// TwinCAT 3 PLC project MonetRoofTests
// Title: MonetRoofTests
// Company: BROT
// ProjectVersion: 0.1.0
// ProgramVersion: 3.1.4024.66
// libraries:
//   MONET Roof, * (Georg-August-Universitaet Goettingen)
//   BROTLib, * (BROT)
//   Tc2_Standard, * (Beckhoff Automation GmbH)
//   Tc2_System, * (Beckhoff Automation GmbH)
//   Tc2_Utilities, * (Beckhoff Automation GmbH)
//   Tc3_Module, * (Beckhoff Automation GmbH)
//   TcUnit, * (www.tcunit.org)
// project tree:
//   / PlcTask.TcTTO
//   POUs/ FB_NullComm.TcPOU, FB_Ramp_Tests.TcPOU, FB_Roof_Consistency_Tests.TcPOU, FB_Roof_State_Tests.TcPOU, MAIN.TcPOU
// real-time tasks:
//   TASK PlcTask: cycle T#10ms, priority 20, ADS port 350

CONFIGURATION MonetRoofTests
    RESOURCE PLC ON TwinCAT3
        TASK PlcTask(INTERVAL := T#10ms, PRIORITY := 20);
        PROGRAM MAIN WITH PlcTask : MAIN;
    END_RESOURCE
END_CONFIGURATION

// ---- POUs/MAIN.TcPOU
PROGRAM MAIN
VAR
	// TcUnit finds every FB_TestSuite instance by itself; it is enough to declare them here.
	fbRampTests				: FB_Ramp_Tests;
	fbRoofConsistencyTests	: FB_Roof_Consistency_Tests;
	fbRoofStateTests		: FB_Roof_State_Tests;
END_VAR

TcUnit.RUN();

END_PROGRAM

// ---- POUs/FB_Ramp_Tests.TcPOU
// Tests for MONETRoof.FB_Ramp, the per-call velocity ramp.
//
// FB_Ramp holds no state of its own: every call recomputes `value` fresh from the `start` input, so
// a multi-cycle ramp only happens because the caller (FB_Roof) feeds its own persisted speed back in
// as `start` each cycle. All these tests can therefore drive a fresh instance directly within a
// single method call, calling it as many times as needed in a FOR loop.
FUNCTION_BLOCK FB_Ramp_Tests EXTENDS TcUnit.FB_TestSuite
VAR
END_VAR

Single_Step_Increases_Toward_Target();
Single_Step_Decreases_Toward_Target();
Reaches_Target_Without_Overshoot();
Reaches_Target_Without_Undershoot();
Large_Reversal_Steps_Instead_Of_Jumping();
Full_Reversal_Ramps_Through_Zero_Over_Many_Cycles();
Zero_Accel_Never_Moves();

METHOD PRIVATE Single_Step_Increases_Toward_Target
VAR
	fbRamp	: MONETRoof.FB_Ramp;
END_VAR
TEST('Single_Step_Increases_Toward_Target');
fbRamp(start := 0, target := 1000, accel := 100);
AssertEquals_INT(Expected := 100, Actual := fbRamp.value, Message := 'one step of 100 towards +1000');
TEST_FINISHED();
END_METHOD

METHOD PRIVATE Single_Step_Decreases_Toward_Target
VAR
	fbRamp	: MONETRoof.FB_Ramp;
END_VAR
TEST('Single_Step_Decreases_Toward_Target');
fbRamp(start := 1000, target := 0, accel := 100);
AssertEquals_INT(Expected := 900, Actual := fbRamp.value, Message := 'one step of 100 towards 0');
TEST_FINISHED();
END_METHOD

METHOD PRIVATE Reaches_Target_Without_Overshoot
VAR
	fbRamp	: MONETRoof.FB_Ramp;
END_VAR
TEST('Reaches_Target_Without_Overshoot');
// 950 + 100 would be 1050: must clamp to the target instead
fbRamp(start := 950, target := 1000, accel := 100);
AssertEquals_INT(Expected := 1000, Actual := fbRamp.value, Message := 'clamped at target, not 1050');
TEST_FINISHED();
END_METHOD

METHOD PRIVATE Reaches_Target_Without_Undershoot
VAR
	fbRamp	: MONETRoof.FB_Ramp;
END_VAR
TEST('Reaches_Target_Without_Undershoot');
// 50 - 100 would be -50: must clamp to the target instead
fbRamp(start := 50, target := 0, accel := 100);
AssertEquals_INT(Expected := 0, Actual := fbRamp.value, Message := 'clamped at target, not -50');
TEST_FINISHED();
END_METHOD

METHOD PRIVATE Large_Reversal_Steps_Instead_Of_Jumping
VAR
	fbRamp	: MONETRoof.FB_Ramp;
END_VAR
// Regression test for code review finding H1: target - value on two INTs overflowed 16 bit for a
// reversal like -30000 -> +30000 (60000 does not fit), which flipped the sign of the comparison and
// jumped straight to the target in one step (fixed by computing it in DINT, FB_Ramp.TcPOU:19-20).
// This asserts one ramp step, not the jump the old code produced.
TEST('Large_Reversal_Steps_Instead_Of_Jumping');
fbRamp(start := -30000, target := 30000, accel := 150);
AssertEquals_INT(Expected := -29850, Actual := fbRamp.value, Message := '-30000 -> +30000: one step of 150, not a jump to +30000');
// symmetric: the same reversal the other way round
fbRamp(start := 30000, target := -30000, accel := 150);
AssertEquals_INT(Expected := 29850, Actual := fbRamp.value, Message := '+30000 -> -30000: one step of 150, not a jump to -30000');
TEST_FINISHED();
END_METHOD

METHOD PRIVATE Full_Reversal_Ramps_Through_Zero_Over_Many_Cycles
VAR
	fbRamp			: MONETRoof.FB_Ramp;
	i				: INT;
	prevValue		: INT;
	curValue		: INT;
	bAllStepsBounded	: BOOL := TRUE;
	valueAtStep200	: INT;
END_VAR
// Drives a full -30000 -> +30000 reversal the way FB_Roof does (feeding value back in as the next
// call's start) and checks every intermediate step, not just the first one. -30000 + 200*150 = 0
// exactly, so this also confirms the ramp actually passes through zero at a known step, not just
// that the endpoints are right. Uses local flags instead of one assertion per loop iteration: TcUnit
// budgets asserts per suite (256 here), and this alone would be 400 calls.
TEST('Full_Reversal_Ramps_Through_Zero_Over_Many_Cycles');
curValue := -30000;
FOR i := 1 TO 400 DO
	prevValue := curValue;
	fbRamp(start := prevValue, target := 30000, accel := 150);
	curValue := fbRamp.value;
	IF ABS(TO_DINT(curValue) - TO_DINT(prevValue)) > 150 THEN
		bAllStepsBounded := FALSE;
	END_IF
	IF i = 200 THEN
		valueAtStep200 := curValue;
	END_IF
END_FOR
AssertTrue(Condition := bAllStepsBounded, Message := 'no single step exceeded accel (150)');
AssertEquals_INT(Expected := 0, Actual := valueAtStep200, Message := 'passes through exactly 0 at step 200 (-30000 + 200*150)');
AssertEquals_INT(Expected := 30000, Actual := curValue, Message := 'reaches target after 400 steps of 150 (60000 / 150)');
TEST_FINISHED();
END_METHOD

METHOD PRIVATE Zero_Accel_Never_Moves
VAR
	fbRamp	: MONETRoof.FB_Ramp;
END_VAR
// accel = 0 is one of the config_error conditions FB_Roof guards against (M0/L6); documented here as
// what FB_Ramp itself does with it, in isolation: it never reaches the target.
TEST('Zero_Accel_Never_Moves');
fbRamp(start := 100, target := 1000, accel := 0);
AssertEquals_INT(Expected := 100, Actual := fbRamp.value, Message := 'accel = 0: value never leaves start');
TEST_FINISHED();
END_METHOD

END_FUNCTION_BLOCK

// ---- POUs/FB_Roof_Consistency_Tests.TcPOU
// Tests for MONETRoof.FB_Roof's consistency checks: sync_error, overtravel_error, config_error (code
// review findings M1, M7 and L6).
//
// TwinCAT only allows external code to WRITE a VAR_INPUT of another instance; a VAR_OUTPUT (even one
// with no AT clause) is read-only from outside, and a plain VAR (no AT/INPUT/OUTPUT) is not reachable
// at all -- only calling a public METHOD on it is. That shapes what these tests can drive:
//   - motors[i].SetPosition(x) works: it is a public METHOD, called on FB_Roof's private motors array
//     element, and is how FB_Roof itself sets a position on a limit snap.
//   - motors[i].position_open / .position_close cannot be written directly (plain VAR_OUTPUT, no
//     setter) -- so limit_error's positive case (a drive that overran its own switch) is not covered
//     here: it needs position_open, which is only ever set by the opened/closed edge, both AT%I*.
//   - position_valid cannot be written directly either (VAR_OUTPUT PERSISTENT, no setter) -- so
//     overtravel_error's positive case is not covered; the negative case (no overtravel_error while
//     position_valid is FALSE, its default) is, since that only needs a read.
// Validate limit_error and overtravel_error's positive cases on the real roof, or with I/O linked in
// a project that has it (MONETN, MONETS) -- same limitation as FB_Roof_State_Tests' opened/closed.
//
// comm is BROTLib.I_Comm, not the roof interface: an unassigned (null) reference would fault the PLC
// the first time an error/state edge tries to log through it, so every roof instance below is given
// an FB_NullComm.
FUNCTION_BLOCK FB_Roof_Consistency_Tests EXTENDS TcUnit.FB_TestSuite
VAR
END_VAR

Sync_Error_When_Positions_Differ_By_Threshold_Or_More();
Sync_Error_Clears_When_Positions_Converge();
No_Overtravel_Error_When_Position_Not_Valid();
Config_Error_When_Max_Position_Not_Above_Min();
Config_Error_When_Speed_Invalid();
Config_Error_Holds_Roof_At_Zero_Speed();

// Shared call with fixed speed/position parameters (10000/30000/150, 0..200), only max_position_diff
// varies per test. Tests that need a different min_position/max_position/speed call fbRoof directly.
METHOD PRIVATE Call
VAR_IN_OUT
	roof		: MONETRoof.FB_Roof;
END_VAR
VAR_INPUT
	comm		: BROTLib.I_Comm;
	maxPosDiff	: INT := 2;
END_VAR
roof(
	roof_number			:= 1,
	min_speed			:= 10000,
	max_speed			:= 30000,
	acceleration		:= 150,
	min_position		:= 0,
	max_position		:= 200,
	max_position_diff	:= maxPosDiff,
	comm				:= comm);
END_METHOD

METHOD PRIVATE Sync_Error_When_Positions_Differ_By_Threshold_Or_More
VAR
	fbRoof	: MONETRoof.FB_Roof;
	fbComm	: FB_NullComm;
END_VAR
TEST('Sync_Error_When_Positions_Differ_By_Threshold_Or_More');
Call(roof := fbRoof, comm := fbComm, maxPosDiff := 2);
AssertFalse(Condition := fbRoof.sync_error, Message := 'both motors start at position 0: in sync');
fbRoof.motors[1].SetPosition(100);
fbRoof.motors[2].SetPosition(102);
Call(roof := fbRoof, comm := fbComm, maxPosDiff := 2);
AssertTrue(Condition := fbRoof.sync_error, Message := 'a difference of 2 (>= max_position_diff) trips sync_error');
TEST_FINISHED();
END_METHOD

METHOD PRIVATE Sync_Error_Clears_When_Positions_Converge
VAR
	fbRoof	: MONETRoof.FB_Roof;
	fbComm	: FB_NullComm;
END_VAR
TEST('Sync_Error_Clears_When_Positions_Converge');
Call(roof := fbRoof, comm := fbComm, maxPosDiff := 2);
fbRoof.motors[1].SetPosition(100);
fbRoof.motors[2].SetPosition(101);
Call(roof := fbRoof, comm := fbComm, maxPosDiff := 2);
AssertFalse(Condition := fbRoof.sync_error, Message := 'a difference of 1 stays below the threshold of 2');
TEST_FINISHED();
END_METHOD

METHOD PRIVATE No_Overtravel_Error_When_Position_Not_Valid
VAR
	fbRoof	: MONETRoof.FB_Roof;
	fbComm	: FB_NullComm;
END_VAR
// M7: position_valid is forced FALSE on the very first cycle and only a limit snap sets it TRUE
// again, so a fresh/unconfirmed position must not arm overtravel_error even when it is wildly off.
TEST('No_Overtravel_Error_When_Position_Not_Valid');
Call(roof := fbRoof, comm := fbComm, maxPosDiff := 2);
AssertFalse(Condition := fbRoof.position_valid, Message := 'position_valid starts FALSE: never confirmed by a limit snap');
fbRoof.Open();
Call(roof := fbRoof, comm := fbComm, maxPosDiff := 2);
fbRoof.motors[1].SetPosition(500);
Call(roof := fbRoof, comm := fbComm, maxPosDiff := 2);
AssertFalse(Condition := fbRoof.overtravel_error, Message := 'no overtravel_error without position_valid, however far off the position is');
TEST_FINISHED();
END_METHOD

METHOD PRIVATE Config_Error_When_Max_Position_Not_Above_Min
VAR
	fbRoof	: MONETRoof.FB_Roof;
	fbComm	: FB_NullComm;
END_VAR
TEST('Config_Error_When_Max_Position_Not_Above_Min');
fbRoof(roof_number := 1, min_speed := 10000, max_speed := 30000, acceleration := 150,
	min_position := 100, max_position := 100, max_position_diff := 2, comm := fbComm);
AssertTrue(Condition := fbRoof.config_error, Message := 'max_position (100) not above min_position (100)');
AssertTrue(Condition := fbRoof.state = E_RoofState.error, Message := 'config_error puts the roof into the error state');
TEST_FINISHED();
END_METHOD

METHOD PRIVATE Config_Error_When_Speed_Invalid
VAR
	fbRoof	: MONETRoof.FB_Roof;
	fbComm	: FB_NullComm;
END_VAR
TEST('Config_Error_When_Speed_Invalid');
fbRoof(roof_number := 1, min_speed := 30000, max_speed := 10000, acceleration := 150,
	min_position := 0, max_position := 200, max_position_diff := 2, comm := fbComm);
AssertTrue(Condition := fbRoof.config_error, Message := 'min_speed (30000) above max_speed (10000)');
TEST_FINISHED();
END_METHOD

METHOD PRIVATE Config_Error_Holds_Roof_At_Zero_Speed
VAR
	fbRoof	: MONETRoof.FB_Roof;
	fbComm	: FB_NullComm;
END_VAR
// L1/config_error interaction: a roof already moving that picks up an invalid parameter (e.g. a
// max_speed above 32767, which would wrap TO_INT and could reverse the direction) must be held at
// zero immediately, unconditionally -- not just flagged.
TEST('Config_Error_Holds_Roof_At_Zero_Speed');
Call(roof := fbRoof, comm := fbComm, maxPosDiff := 2);
fbRoof.Open();
Call(roof := fbRoof, comm := fbComm, maxPosDiff := 2);
AssertFalse(Condition := fbRoof.config_error, Message := 'valid parameters so far');
fbRoof(roof_number := 1, min_speed := 10000, max_speed := 40000, acceleration := 150,
	min_position := 0, max_position := 200, max_position_diff := 2, comm := fbComm);
AssertTrue(Condition := fbRoof.config_error, Message := 'max_speed above 32767 wraps TO_INT: config_error catches it');
AssertTrue(Condition := fbRoof.state = E_RoofState.error, Message := 'error state; drive held, slow mode included (FB_Roof.TcPOU config_error stop)');
TEST_FINISHED();
END_METHOD

END_FUNCTION_BLOCK

// ---- POUs/FB_NullComm.TcPOU
// No-op I_Comm implementation for tests. FB_Roof/FB_RoofMotor call Comm.Publish / Comm.PublishLog
// (via FB_EventLog) on error/state edges; a null (unassigned) I_Comm reference there would fault the
// PLC, so every FB_Roof test instance is given one of these instead of a real MQTT connection.
FUNCTION_BLOCK FB_NullComm IMPLEMENTS BROTLib.I_Comm
VAR
	// number of Publish/PublishLog calls seen, in case a test ever wants to assert an event fired
	nPublishCalls		: UDINT;
	nPublishLogCalls	: UDINT;
END_VAR

METHOD Publish : BOOL
VAR_INPUT
	domain			: STRING(255) := 'environment';
	location		: STRING(255) := 'roof';
	parameter		: STRING(255);
	value			: STRING(255);
END_VAR
VAR_OUTPUT
	published	: BOOL;
END_VAR
nPublishCalls := nPublishCalls + 1;
published := TRUE;
Publish := TRUE;
END_METHOD

METHOD PublishLog : BOOL
VAR_INPUT
	level		: STRING(255) := 'INFO';
	message		: STRING(255);
END_VAR
VAR_OUTPUT
	published	: BOOL;
END_VAR
nPublishLogCalls := nPublishLogCalls + 1;
published := TRUE;
PublishLog := TRUE;
END_METHOD

END_FUNCTION_BLOCK

// ---- POUs/FB_Roof_State_Tests.TcPOU
// Tests for MONETRoof.FB_Roof's state machine (code review finding L5): the E_RoofState.unknown default
// before the first call, and what the roof does while a drive reports an error.
//
// In this project every drive reports an error: FB_RoofMotor.motor_error is AT%I* and means "drive OK"
// (error := NOT motor_error), and no I/O is mapped here, so it stays FALSE. FB_Roof therefore sits in the
// error state from its first call. A test cannot set motor_error from outside (it is a VAR_OUTPUT of an
// internal variable; TwinCAT only accepts assignments to inputs). The transitions that need healthy drives
// (stopped, opening, closing, opened, closed, and Reset() clearing the latched error once the fault is
// gone) are therefore validated on the PLC with the real hardware, like the plan's open step 5.
FUNCTION_BLOCK FB_Roof_State_Tests EXTENDS TcUnit.FB_TestSuite
VAR
END_VAR

Initial_State_Is_Unknown();
Drive_Error_Puts_Roof_In_Error_State();
Open_Is_Refused_While_Drive_Error();
Close_Is_Refused_While_Drive_Error();
Reset_Does_Not_Clear_A_Drive_Error();

METHOD PRIVATE Call
VAR_IN_OUT
	roof		: MONETRoof.FB_Roof;
END_VAR
VAR_INPUT
	comm		: BROTLib.I_Comm;
END_VAR
roof(
	roof_number			:= 1,
	min_speed			:= 10000,
	max_speed			:= 30000,
	acceleration		:= 150,
	min_position		:= 0,
	max_position		:= 200,
	max_position_diff	:= 2,
	comm				:= comm);
END_METHOD

METHOD PRIVATE Initial_State_Is_Unknown
VAR
	fbRoof	: MONETRoof.FB_Roof;
END_VAR
// Before FB_Roof is ever called, its VAR_OUTPUT members already hold their declared defaults.
TEST('Initial_State_Is_Unknown');
AssertTrue(Condition := fbRoof.state = E_RoofState.unknown, Message := 'declared default before the first call (was closed / enum value 0, L5)');
TEST_FINISHED();
END_METHOD

METHOD PRIVATE Open_Is_Refused_While_Drive_Error
VAR
	fbRoof	: MONETRoof.FB_Roof;
	fbComm	: FB_NullComm;
END_VAR
TEST('Open_Is_Refused_While_Drive_Error');
Call(roof := fbRoof, comm := fbComm);	// assigns the parameters; Open() before this would see max_speed = 0
fbRoof.Open();
Call(roof := fbRoof, comm := fbComm);
AssertTrue(Condition := fbRoof.state = E_RoofState.error, Message := 'Open() with a drive error: the error stop wins, the roof never reaches opening');
TEST_FINISHED();
END_METHOD

METHOD PRIVATE Drive_Error_Puts_Roof_In_Error_State
VAR
	fbRoof	: MONETRoof.FB_Roof;
	fbComm	: FB_NullComm;
END_VAR
TEST('Drive_Error_Puts_Roof_In_Error_State');
Call(roof := fbRoof, comm := fbComm);
AssertTrue(Condition := fbRoof.state = E_RoofState.error, Message := 'motor_error is FALSE (no I/O): both drives report an error, so the roof is in the error state');
TEST_FINISHED();
END_METHOD

METHOD PRIVATE Close_Is_Refused_While_Drive_Error
VAR
	fbRoof	: MONETRoof.FB_Roof;
	fbComm	: FB_NullComm;
END_VAR
TEST('Close_Is_Refused_While_Drive_Error');
Call(roof := fbRoof, comm := fbComm);	// assigns the parameters
fbRoof.Close();
Call(roof := fbRoof, comm := fbComm);
AssertTrue(Condition := fbRoof.state = E_RoofState.error, Message := 'Close() with a drive error: the error stop wins, the roof never reaches closing');
TEST_FINISHED();
END_METHOD

METHOD PRIVATE Reset_Does_Not_Clear_A_Drive_Error
VAR
	fbRoof	: MONETRoof.FB_Roof;
	fbComm	: FB_NullComm;
END_VAR
TEST('Reset_Does_Not_Clear_A_Drive_Error');
// invalid parameters (max_position = min_position) force config_error and the error state
fbRoof(roof_number := 1, min_speed := 10000, max_speed := 30000, acceleration := 150,
	min_position := 100, max_position := 100, max_position_diff := 2, comm := fbComm);
AssertTrue(Condition := fbRoof.config_error, Message := 'sanity: invalid parameters set config_error');
fbRoof.Reset();
// valid parameters now, reset_roof is pending: the parameter fault is gone, the drive error is not
Call(roof := fbRoof, comm := fbComm);
AssertFalse(Condition := fbRoof.config_error, Message := 'valid parameters now');
AssertTrue(Condition := fbRoof.state = E_RoofState.error, Message := 'a reset must not hide a drive error that is still present');
TEST_FINISHED();
END_METHOD

END_FUNCTION_BLOCK
